TYPE E_OdriveControlMode :
(
    Voltage := 0,
    Torque := 1,
    Velocity := 2,
    Position := 3
) UDINT;
END_TYPE

(* stored: Version 1.1.0.1
   DUT E_OdriveControlMode: Id {359d4e0e-21e9-4560-8ed9-483f3e9ca3da} *)
